// LS Electric XG5000 project: 2021년 지방과제
// PLC NewPLC
// module base 0 slot 0: 입출력 모듈:XBC-DR32H (DC 24V 입력, 릴레이 출력 32점)
// module base 0 slot 1: 위치결정 모듈:XBF-PD02A (위치결정 펄스(LD)출력형, 2축)
// module base 0 slot 2: 출력 모듈:XBE-TN/TP16A (트랜지스터 출력, 16점 (싱크출력/소스출력))

PROGRAM NewProgram (task: 스캔 프로그램)

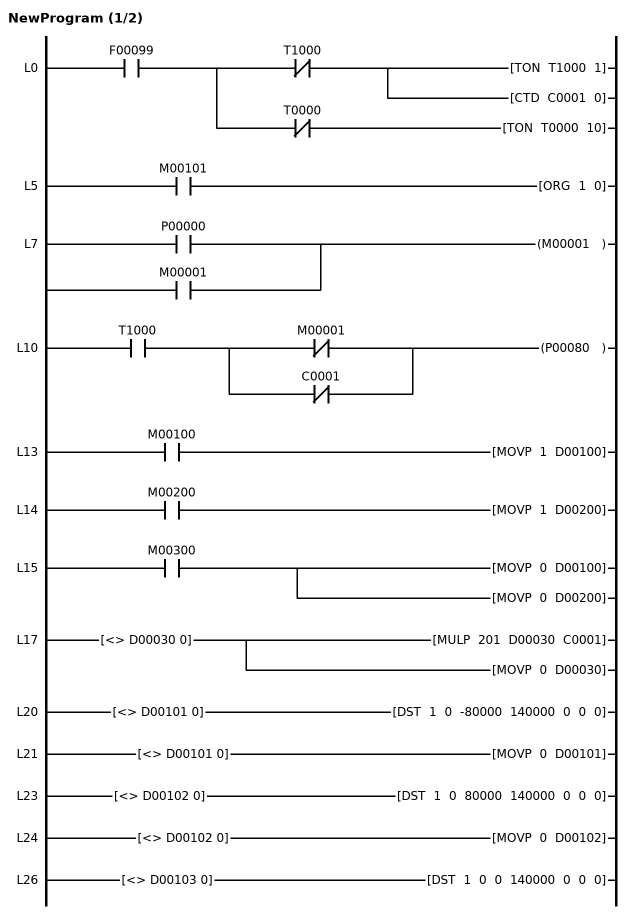
; L0
LOAD      F00099
MPUSH
AND NOT   T1000
TON       T1000 1
CTD       C0001 0
MPOP
AND NOT   T0000
TON       T0000 10
; L5
LOAD      M00101
ORG       1 0
; L7
LOAD      P00000
OR        M00001
OUT       M00001
; L10
LOAD      T1000
LOAD NOT  M00001
OR NOT    C0001
AND LOAD
OUT       P00080
; L13
LOAD      M00100
MOVP      1 D00100
; L14
LOAD      M00200
MOVP      1 D00200
; L15
LOAD      M00300
MOVP      0 D00100
MOVP      0 D00200
; L17
LOAD<>    D00030 0
MULP      201 D00030 C0001
MOVP      0 D00030
; L20
LOAD<>    D00101 0
DST       1 0 -80000 140000 0 0 0
; L21
LOAD<>    D00101 0
MOVP      0 D00101
; L23
LOAD<>    D00102 0
DST       1 0 80000 140000 0 0 0
; L24
LOAD<>    D00102 0
MOVP      0 D00102
; L26
LOAD<>    D00103 0
DST       1 0 0 140000 0 0 0

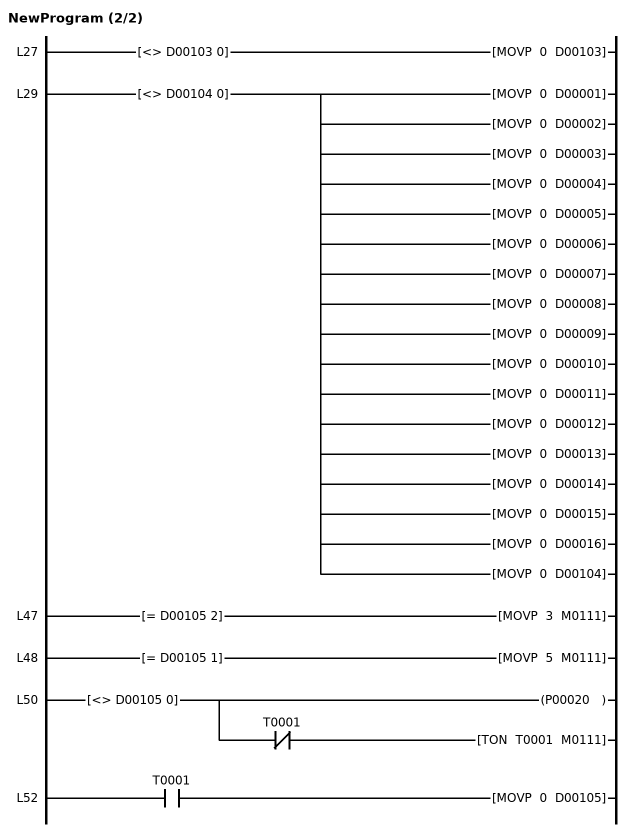
; L27
LOAD<>    D00103 0
MOVP      0 D00103
; L29
LOAD<>    D00104 0
MOVP      0 D00001
MOVP      0 D00002
MOVP      0 D00003
MOVP      0 D00004
MOVP      0 D00005
MOVP      0 D00006
MOVP      0 D00007
MOVP      0 D00008
MOVP      0 D00009
MOVP      0 D00010
MOVP      0 D00011
MOVP      0 D00012
MOVP      0 D00013
MOVP      0 D00014
MOVP      0 D00015
MOVP      0 D00016
MOVP      0 D00104
; L47
LOAD=     D00105 2
MOVP      3 M0111
; L48
LOAD=     D00105 1
MOVP      5 M0111
; L50
LOAD<>    D00105 0
OUT       P00020
AND NOT   T0001
TON       T0001 M0111
; L52
LOAD      T0001
MOVP      0 D00105

VARIABLES AND COMMENTS (devices not used above)
M01000	BIT	PB0